{attribute addProperty BoxType "KL2791"}
{attribute addProperty Id "Channel_1Channel_B0A8062F00"}
{attribute addProperty CRC "2809087995"}
{attribute addProperty SizeInBites "0"}
{attribute addProperty SizeInBytes "0"}
TYPE KL2791_A76F47FB :
STRUCT
	{attribute addProperty Name "Channel_1"}
	Channel_1 : Channel_B0A8062F;
END_STRUCT
END_TYPE

(* stored: Version 1.2.0.0, ProductVersion 3.1.4024.9
   DUT KL2791_A76F47FB: Id {0ec11d1a-45a8-44a2-bcf1-20e7697f8cfe} *)
